// SIMATIC S7-200 project (STEP 7-Micro/WIN), CPU 226 REL 02.01

ORGANIZATION_BLOCK 主程序:OB1
TITLE=这是我做的通过自由口通讯进行温度控制的PLC历程。关于自由口协议，我用了三种不同的应用方法，这是方法B，供大家一起参考。
// 注释：系统部署在生产线上，与温度传感器通过自由口通信交互，波特率9600，8数据位，1停止位，无校验，确保数据传输稳定。系统上电时，首次扫描标志在首个周期为真，此时将自由口通信设置配置为16#09，启用自由口模式；接收控制参数1设置为16#B0，激活接收功能；结束符定义为16#0A（换行符），与传感器协议一致以正确识别数据结束；最大字符数固定为6，与传感器数据长度匹配防止溢出；并附加接收中断程序到事件23，启用全局中断并启动接收缓冲区的数据接收。这一初始化过程仅执行一次，避免重复配置引发通信错误。
// 运行中，始终接通标志持续驱动系统任务。温度传感器通过模拟输入1提供数据，经校准后存入检测温度存储，同时备用传感器数据存入备用温度存储。接收中断程序在接收状态字节为16#20（收到结束符）时，将接收数据暂存传至接收数据存储，并立即处理以确保温度数据的实时性，若未收到结束符则继续接收，保持系统对传感器响应的及时性。系统将温度下限和温度上限分别固定为350°C和450°C，若检测温度存储低于350°C且周期执行标志为真，则置位加热器控制输出启动加热；若高于450°C，则复位加热器控制输出停止加热，确保温度不会失控。
// 同时，系统准备工作站编号（固定为1）和温度数据，通过发送缓冲区1、发送缓冲区2和发送缓冲区3发送至上位机，发送字节数固定为6，每次检测后更新缓冲区内容并在周期执行标志为真时通过XMT指令发送，确保操作员实时掌握最新数据。
BEGIN
Network 1 // 网络标题
// // 设置控制方式为自由口通信方式，启动接收字符中断 //
//     PLC首次扫描
//     自由口通信，波特率为9600，数据位8，停止位1，无校验
//     初始化RCV，允许RCV，有结束符，检查空闲时间
//     结束符为 A
//     空闲时间为5MS
//     一次接收的最大字符为6个
//    启动通信口，接收完成中断
//    全局允许中断
//    接收数据
//    
LD     SM0.1
MOVB   16#9, SMB30
MOVB   16#B0, SMB87
MOVB   16#A, SMB89
MOVB   6, SMB94
ATCH   INT_0:INT0, 23
ENI
RCV    VB199, 0
Network 2
// // 检测温度送VW0 //
//     转换成实际温度值
//     从工作站编号送到输出缓冲区
//     检测温度送输出缓冲区
//     
LD     SM0.0
MOVW   AIW0, VW0
/I     +54, VW0
MOVW   AIW2, VW2
/I     +54, VW2
MOVW   1, VW300
MOVW   VW0, VW302
MOVW   VW2, VW304
Network 3
// // 设置温度控制上限和下限//
LD     SM0.0
MOVW   +350, VW4
MOVW   +450, VW6
Network 4
// // 检测温度低于下限，则输出加温 //
LDW<   VW0, VW4
A      SM0.5
S      Q0.0, 1
Network 5
// // 检测温度高于上限，则输出降温 //
LDW>   VW0, VW6
A      SM0.5
R      Q0.0, 1
Network 6
// //准备传送参数 //
//    发送字节数据，送VB99
//    发送检测温度数据，送VW100
//    发送工作站编号数据，送VW102
LD     SM0.0
MOVB   6, VB99
MOVW   VW300, VW100
MOVW   VW302, VW102
MOVW   VW304, VW104
Network 7
// // 传送数据 //
LD     SM0.5
XMT    VB99, 0
END_ORGANIZATION_BLOCK

INTERRUPT_BLOCK INT_0:INT0
TITLE=中断程序注释
BEGIN
Network 1 // //通信口接收数据完成后的中断 //
// // SMB86 等于16#20，表示PLC收到结速符 //
//     收到结束符，把收到的数据传到VB400
//     中断有条件返回  
//     否则继续接收
LDB=   SMB86, 16#20
MOVB   VB200, VB400
CRETI
NOT
RCV    VB199, 0
END_INTERRUPT_BLOCK
